// TIA Portal V17 export
// export: Created 2024-08-09T12:53:19.8649511Z, ExportSetting WithDefaults, DisplayName Totally Integrated Automation Portal, DisplayVersion V17 Update 7, DisplayName TIA Portal Openness, DisplayVersion V17 Update 7, DisplayName TIA Portal Version Control Interface, DisplayVersion V17, DisplayName STEP 7 Professional, DisplayVersion V17 Update 7, DisplayName STEP 7 Safety, DisplayVersion V17 Update 6, DisplayName WinCC Professional, DisplayVersion V17 Update 7
TYPE "S_Data_Reception"
// stored: IsFailsafeCompliant false
   STRUCT
      Densite : Real := 0.0;   // Densite matiere
      DensiteInit : Real := 0.0;   // Densit initiale de la matire réceptionne
      QteTheo : Real := 0.0;   // Quantité théorique a receptionner
      QteReel : Real := 0.0;   // Quantit reel calcule ;passe sur le transporteur
      Debit : Real := 0.0;   // Débit massique transporteur
      QtePossibleCellule : Real := 0.0;   // Quantité possible dans la cellule de destination
      TpsDepuis : Int := 0;   // Temps de transfert sur le transporteur
      TpsReste : Int := 0;
      Fg_Aff_bt_Acq_Nett : Int := 0;   // Affichage du bouton d'acquit fosse propre sur supervision
      CdMat : String["T_CD_MAT"];
      Origine : String["T_CD_CEL"];
      Dest : String["T_CD_CEL"];
      Dest2 : String["T_CD_CEL"];
      Dest3 : String["T_CD_CEL"];
      No_LotF : String;   // Numro de lot associé a la matière stocke
      Cd_Rec : String["T_CD_REC"];
      Cd_Badge : String[20];   // No de badge envoyé a la base de donne (si lancement avec badge)
   END_STRUCT;
END_TYPE
